// TIA Portal project "THESIS SCADA" (V15)

(* hardware
DEVICE "PC-System_1"  SIMATIC PC station
   slot 0: "SIMATIC PC station"  Rail  SIMATIC PC-Station  V1.0
      slot 125: "Stationmanager"  Station_Manager  V6.0.4
   slot 1: "HMI_RT_1"  WinCC RT Advanced  6AV2 104-0xxxx-xxxx  15.0.0.0
      slot 33792: "Host interface"  Host interface
*)

(* ===== HMI "HMI_RT_1" =====
system functions are stored by id; their names below are inferred from use
connection "Connection_1": OPC, OPC

HMI tags "Default tag table"
   "E1ALARM" : VT_I2, 1 s
   "E2ALARM" : VT_I2, 1 s
   "E3ALARM" : VT_I2, 1 s
   "E4ALARM" : VT_I2, 1 s
   "E1CAR" : VT_BOOL, 1 s
   "E2CAR" : VT_BOOL, 1 s
   "E3CAR" : VT_BOOL, 1 s
   "E4CAR" : VT_BOOL, 1 s
   "H0UP" : VT_BOOL, 1 s
   "H0DOWN" : VT_BOOL, 1 s
   "H1UP" : VT_BOOL, 1 s
   "H1DOWN" : VT_BOOL, 1 s
   "H2UP" : VT_BOOL, 1 s
   "H2DOWN" : VT_BOOL, 1 s
   "H3UP" : VT_BOOL, 1 s
   "H3DOWN" : VT_BOOL, 1 s
   "H4UP" : VT_BOOL, 1 s
   "H4DOWN" : VT_BOOL, 1 s
   "H5UP" : VT_BOOL, 1 s
   "H5DOWN" : VT_BOOL, 1 s
   "H6UP" : VT_BOOL, 1 s
   "H6DOWN" : VT_BOOL, 1 s
   "H7UP" : VT_BOOL, 1 s
   "H7DOWN" : VT_BOOL, 1 s
   "H8UP" : VT_BOOL, 1 s
   "H8DOWN" : VT_BOOL, 1 s
   "H9UP" : VT_BOOL, 1 s
   "H9DOWN" : VT_BOOL, 1 s
   "H10UP" : VT_BOOL, 1 s
   "H10DOWN" : VT_BOOL, 1 s
   "H11UP" : VT_BOOL, 1 s
   "H11DOWN" : VT_BOOL, 1 s
   "H12UP" : VT_BOOL, 1 s
   "H12DOWN" : VT_BOOL, 1 s
   "H13UP" : VT_BOOL, 1 s
   "H13DOWN" : VT_BOOL, 1 s
   "H14UP" : VT_BOOL, 1 s
   "H14DOWN" : VT_BOOL, 1 s
   "H15UP" : VT_BOOL, 1 s
   "H16DOWN" : VT_BOOL, 1 s
   "H17UP" : VT_BOOL, 1 s
   "H17DOWN" : VT_BOOL, 1 s
   "H18UP" : VT_BOOL, 1 s
   "H18DOWN" : VT_BOOL, 1 s
   "H19UP" : VT_BOOL, 1 s
   "H19DOWN" : VT_BOOL, 1 s
   "E1FLOOR0" : VT_BOOL, 1 s
   "E1FLOOR1" : VT_BOOL, 1 s
   "E1FLOOR2" : VT_BOOL, 1 s
   "E1FLOOR3" : VT_BOOL, 1 s
   "E1FLOOR4" : VT_BOOL, 1 s
   "E1FLOOR5" : VT_BOOL, 1 s
   "E1FLOOR6" : VT_BOOL, 1 s
   "E1FLOOR7" : VT_BOOL, 1 s
   "E1FLOOR8" : VT_BOOL, 1 s
   "E1FLOOR9" : VT_BOOL, 1 s
   "E1FLOOR10" : VT_BOOL, 1 s
   "E1FLOOR11" : VT_BOOL, 1 s
   "E1FLOOR12" : VT_BOOL, 1 s
   "E1FLOOR13" : VT_BOOL, 1 s
   "E2FLOOR0" : VT_BOOL, 1 s
   "E2FLOOR1" : VT_BOOL, 1 s
   "E2FLOOR2" : VT_BOOL, 1 s
   "E2FLOOR3" : VT_BOOL, 1 s
   "E2FLOOR4" : VT_BOOL, 1 s
   "E2FLOOR5" : VT_BOOL, 1 s
   "E2FLOOR6" : VT_BOOL, 1 s
   "E2FLOOR7" : VT_BOOL, 1 s
   "E2FLOOR8" : VT_BOOL, 1 s
   "E2FLOOR9" : VT_BOOL, 1 s
   "E2FLOOR10" : VT_BOOL, 1 s
   "E2FLOOR11" : VT_BOOL, 1 s
   "E2FLOOR12" : VT_BOOL, 1 s
   "E2FLOOR13" : VT_BOOL, 1 s
   "E3FLOOR0" : VT_BOOL, 1 s
   "E3FLOOR1" : VT_BOOL, 1 s
   "E3FLOOR2" : VT_BOOL, 1 s
   "E3FLOOR3" : VT_BOOL, 1 s
   "E3FLOOR4" : VT_BOOL, 1 s
   "E3FLOOR5" : VT_BOOL, 1 s
   "E3FLOOR6" : VT_BOOL, 1 s
   "E3FLOOR7" : VT_BOOL, 1 s
   "E3FLOOR8" : VT_BOOL, 1 s
   "E3FLOOR9" : VT_BOOL, 1 s
   "E3FLOOR10" : VT_BOOL, 1 s
   "E3FLOOR11" : VT_BOOL, 1 s
   "E3FLOOR12" : VT_BOOL, 1 s
   "E3FLOOR13" : VT_BOOL, 1 s
   "E4FLOOR5" : VT_BOOL, 1 s
   "E4FLOOR6" : VT_BOOL, 1 s
   "E4FLOOR7" : VT_BOOL, 1 s
   "E4FLOOR8" : VT_BOOL, 1 s
   "E4FLOOR9" : VT_BOOL, 1 s
   "E4FLOOR10" : VT_BOOL, 1 s
   "E4FLOOR11" : VT_BOOL, 1 s
   "E4FLOOR12" : VT_BOOL, 1 s
   "E4FLOOR13" : VT_BOOL, 1 s
   "E4FLOOR14" : VT_BOOL, 1 s
   "E4FLOOR15" : VT_BOOL, 1 s
   "E4FLOOR16" : VT_BOOL, 1 s
   "E4FLOOR17" : VT_BOOL, 1 s
   "E4FLOOR18" : VT_BOOL, 1 s
   "E4FLOOR19" : VT_BOOL, 1 s
   "E1CURRENTFLOOR" : VT_I2, 1 s
   "E2CURRENTFLOOR" : VT_I2, 1 s
   "E3CURRENTFLOOR" : VT_I2, 1 s
   "E4CURRENTFLOOR" : VT_I2, 1 s
   "E1UP" : VT_BOOL, 1 s
   "E1DOWN" : VT_BOOL, 1 s
   "E2UP" : VT_BOOL, 1 s
   "E2DOWN" : VT_BOOL, 1 s
   "E3UP" : VT_BOOL, 1 s
   "E3DOWN" : VT_BOOL, 1 s
   "E4UP" : VT_BOOL, 1 s
   "E4DOWN" : VT_BOOL, 1 s
   "ALARMRESET" : VT_BOOL, 1 s
   "ALARMNOT/RST" : VT_BOOL, 1 s
   "H16UP" : VT_BOOL, 1 s
   "H15DOWN" : VT_BOOL, 1 s
   "e1nextfloor" : VT_I2, 1 s
   "e2nextfloor" : VT_I2, 1 s
   "e3nextfloor" : VT_I2, 1 s
   "e4nextfloor" : VT_I2, 1 s

discrete alarms
   1: 'PLEASE GIVE CARCALL IN RESPECTIVE ELEVATOR DIRECTION', class Errors, trigger "E1ALARM" bit 0
   2: 'PLEASE GIVE CARCALL IN RESPECTIVE ELEVATOR DIRECTION', class Errors, trigger "E2ALARM" bit 0
   3: 'PLEASE GIVE CARCALL IN RESPECTIVE ELEVATOR DIRECTION', class Errors, trigger "E3ALARM" bit 0
   4: 'PLEASE GIVE CARCALL IN RESPECTIVE ELEVATOR DIRECTION', class Errors, trigger "E4ALARM" bit 0

screen "HALLCALL" 800x600
   TextField "Text field_1" at 208,16 size 148x37; Text 'HALLCALL'
   TextField "Text field_22" at 624,8 size 139x28; Text 'NAVIGATION'
   TextField "Text field_23" at 624,96 size 135x22; Text 'CURRENT FLOOR'
   TextField "Text field_24" at 624,208 size 135x22; Text 'CURRENT FLOOR'
   TextField "Text field_25" at 624,320 size 135x22; Text 'CURRENT FLOOR'
   TextField "Text field_26" at 632,432 size 135x22; Text 'CURRENT FLOOR'
   Group "Group_1" at 32,72 size 496x504
   Group "Group_2" at 648,544 size 96x31
   Group "Group_3" at 648,544 size 96x39
   Group "Group_4" at 648,544 size 96x40
   Group "Group_5" at 648,544 size 96x40
   Group "Group_6" at 648,544 size 96x40
   Group "Group_7" at 648,544 size 96x40
   Group "Group_8" at 648,544 size 96x40
   Group "Group_9" at 648,544 size 96x40
   Button "Button_1" at 640,280 size 96x32; TextOff 'E3CAR'
      on Click: ActivateScreen("E3CAR", 0)
   Button "Button_2" at 640,392 size 96x32; TextOff 'E4CAR'
      on Click: ActivateScreen("E4CAR", 0)
   Button "Button_3" at 640,168 size 96x32; TextOff 'E2CAR'
      on Click: ActivateScreen("E2CAR", 0)
   Button "Button_4" at 640,56 size 96x32; TextOff 'E1CAR'
      on Click: ActivateScreen("E1CAR", 0)
      Appearance <- "E1CAR"
   Button "Button_5" at 648,504 size 96x32; TextOff 'ALARM'
      on Click: ActivateScreen("ALARM", 0)
   IOField "I/O field_1" at 672,128 size 40x32; FormatPattern 11
      ProcessValue <- "E1CURRENTFLOOR"
   IOField "I/O field_2" at 672,240 size 40x32; FormatPattern 11
      ProcessValue <- "E2CURRENTFLOOR"
   IOField "I/O field_3" at 672,352 size 40x32; FormatPattern 11
      ProcessValue <- "E3CURRENTFLOOR"
   IOField "I/O field_4" at 672,464 size 40x32; FormatPattern 11
      ProcessValue <- "E4CURRENTFLOOR"
   Button "Button_24" at 48,94 size 96x32; TextOff 'H9UP'
      on Press: SetBit("H9UP")
      Appearance <- "H9UP"
   TextField "Text field_11" at 145,100 size 15x22; Text '9'
   Button "Button_25" at 161,94 size 96x32; TextOff 'H9DOWN'
      on Press: SetBit("H9DOWN")
      Appearance <- "H9DOWN"
   Button "Button_22" at 48,142 size 96x32; TextOff 'H8UP'
      on Press: SetBit("H8UP")
      Appearance <- "H8UP"
   TextField "Text field_10" at 145,148 size 15x22; Text '8'
   Button "Button_23" at 161,142 size 96x32; TextOff 'H8DOWN'
      on Press: SetBit("H8DOWN")
      Appearance <- "H8DOWN"
   Button "Button_20" at 48,190 size 96x32; TextOff 'H7UP'
      on Press: SetBit("H7UP")
      Appearance <- "H7UP"
   TextField "Text field_9" at 145,196 size 15x22; Text '7'
   Button "Button_21" at 161,190 size 96x32; TextOff 'H7DOWN'
      on Press: SetBit("H7DOWN")
      Appearance <- "H7DOWN"
   Button "Button_18" at 48,238 size 96x32; TextOff 'H6UP'
      on Press: SetBit("H6UP")
      Appearance <- "H6UP"
   TextField "Text field_8" at 145,244 size 15x22; Text '6'
   Button "Button_19" at 161,238 size 96x32; TextOff 'H6DOWN'
      on Press: SetBit("H6DOWN")
      Appearance <- "H0DOWN"
   Button "Button_16" at 48,286 size 96x32; TextOff 'H5UP'
      on Press: SetBit("H5UP")
      Appearance <- "H5UP"
   TextField "Text field_7" at 145,292 size 15x22; Text '5'
   Button "Button_17" at 161,286 size 96x32; TextOff 'H5DOWN'
      on Press: SetBit("H5DOWN")
      Appearance <- "H5DOWN"
   Button "Button_14" at 48,334 size 96x32; TextOff 'H4UP'
      on Press: SetBit("H4UP")
      Appearance <- "H4UP"
   TextField "Text field_6" at 145,340 size 15x22; Text '4'
   Button "Button_15" at 161,334 size 96x32; TextOff 'H4DOWN'
      on Press: SetBit("H4DOWN")
      Appearance <- "H4DOWN"
   Button "Button_12" at 48,382 size 96x32; TextOff 'H3UP'
      on Press: SetBit("H3UP")
      Appearance <- "H3UP"
   TextField "Text field_5" at 145,388 size 15x22; Text '3'
   Button "Button_13" at 161,382 size 96x32; TextOff 'H3DOWN'
      on Press: SetBit("H3DOWN")
      Appearance <- "H3DOWN"
   Button "Button_10" at 48,430 size 96x32; TextOff 'H2UP'
      on Press: SetBit("H2UP")
      Appearance <- "H2UP"
   TextField "Text field_4" at 145,436 size 15x22; Text '2'
   Button "Button_11" at 161,430 size 96x32; TextOff 'H2DOWN'
      on Press: SetBit("H2DOWN")
      Appearance <- "H2DOWN"
   Button "Button_8" at 48,478 size 96x32; TextOff 'H1UP'
      on Press: SetBit("H1UP")
      Appearance <- "H1UP"
   TextField "Text field_3" at 145,484 size 15x22; Text '1'
   Button "Button_9" at 161,478 size 96x32; TextOff 'H1DOWN'
      on Press: SetBit("H1DOWN")
      Appearance <- "H1DOWN"
   Button "Button_6" at 48,526 size 96x32; TextOff 'H0UP'
      on Press: SetBit("H0UP")
      Appearance <- "H0UP"
   TextField "Text field_2" at 145,532 size 15x22; Text '0'
   Button "Button_7" at 161,526 size 96x32; TextOff 'H0DOWN'
      on Press: SetBit("H0DOWN")
      Appearance <- "H0DOWN"
   Button "Button_44" at 288,94 size 96x32; TextOff 'H19UP'
      on Press: SetBit("H19UP")
      Appearance <- "H19UP"
   TextField "Text field_21" at 385,100 size 25x22; Text '19'
   Button "Button_45" at 410,93 size 96x32; TextOff 'H19DOWN'
      on Press: SetBit("H19DOWN")
      Appearance <- "H19DOWN"
   Button "Button_42" at 288,142 size 96x32; TextOff 'H18UP'
      on Press: SetBit("H18UP")
      Appearance <- "H18UP"
   TextField "Text field_20" at 385,148 size 25x22; Text '18'
   Button "Button_43" at 410,141 size 96x32; TextOff 'H18DOWN'
      on Press: SetBit("H18DOWN")
      Appearance <- "H18DOWN"
   Button "Button_40" at 288,190 size 96x32; TextOff 'H17UP'
      on Press: SetBit("H17UP")
      Appearance <- "H17UP"
   TextField "Text field_19" at 385,196 size 25x22; Text '17'
   Button "Button_41" at 410,189 size 96x32; TextOff 'H17DOWN'
      on Press: SetBit("H17DOWN")
      Appearance <- "H17DOWN"
   Button "Button_38" at 288,238 size 96x32; TextOff 'H16UP'
      on Press: SetBit("H16UP")
      Appearance <- "H16UP"
   TextField "Text field_18" at 385,244 size 25x22; Text '16'
   Button "Button_39" at 410,237 size 96x32; TextOff 'H16DOWN'
      on Press: SetBit("H16DOWN")
      Appearance <- "H16DOWN"
   Button "Button_36" at 288,286 size 96x32; TextOff 'H15UP'
      on Press: SetBit("H15UP")
      Appearance <- "H15UP"
   TextField "Text field_17" at 385,292 size 25x22; Text '15'
   Button "Button_37" at 410,285 size 96x32; TextOff 'H15DOWN'
      on Press: SetBit("H15DOWN")
      Appearance <- "H15DOWN"
   Button "Button_34" at 288,334 size 96x32; TextOff 'H14UP'
      on Press: SetBit("H14UP")
      Appearance <- "H14UP"
   TextField "Text field_16" at 385,340 size 25x22; Text '14'
   Button "Button_35" at 410,333 size 96x32; TextOff 'H14DOWN'
      on Press: SetBit("H14DOWN")
      Appearance <- "H14DOWN"
   Button "Button_32" at 288,382 size 96x32; TextOff 'H13UP'
      on Press: SetBit("H13UP")
      Appearance <- "H13UP"
   TextField "Text field_15" at 385,388 size 25x22; Text '13'
   Button "Button_33" at 410,381 size 96x32; TextOff 'H13DOWN'
      on Press: SetBit("H13DOWN")
      Appearance <- "H13DOWN"
   Button "Button_30" at 288,430 size 96x32; TextOff 'H12UP'
      on Press: SetBit("H12UP")
      Appearance <- "H12UP"
   TextField "Text field_14" at 385,436 size 25x22; Text '12'
   Button "Button_31" at 410,429 size 96x32; TextOff 'H12DOWN'
      on Press: SetBit("H12DOWN")
      Appearance <- "H12DOWN"
   Button "Button_28" at 288,478 size 96x32; TextOff 'H11UP'
      on Press: SetBit("H11UP")
      Appearance <- "H11UP"
   TextField "Text field_13" at 385,484 size 25x22; Text '11'
   Button "Button_29" at 410,477 size 96x32; TextOff 'H11DOWN'
      on Press: SetBit("H11DOWN")
      Appearance <- "H11DOWN"
   Button "Button_26" at 288,526 size 96x32; TextOff 'H10UP'
      on Press: SetBit("H10UP")
      Appearance <- "H10UP"
   TextField "Text field_12" at 385,532 size 25x22; Text '10'
   Button "Button_27" at 410,525 size 96x32; TextOff 'H10DOWN'
      on Press: SetBit("H10DOWN")
      Appearance <- "H10DOWN"
   TextField "Text field_27" at 651,552 size 86x22; Text 'NO ALARM'
   Rectangle "Rectangle_24" at 648,544 size 96x39
      Visibility <- "E4ALARM"
   TextField "Text field_28" at 655,555 size 81x22; Text 'E4 ALARM'
      Visibility <- "E4ALARM"
   TextField "Text field_29" at 651,554 size 86x22; Text 'NO ALARM'
   Rectangle "Rectangle_26" at 648,544 size 96x40
      Visibility <- "E3ALARM"
   TextField "Text field_30" at 655,555 size 81x22; Text 'E3 ALARM'
      Visibility <- "E3ALARM"
   TextField "Text field_31" at 651,554 size 86x22; Text 'NO ALARM'
   Rectangle "Rectangle_28" at 648,544 size 96x40
      Visibility <- "E2ALARM"
   TextField "Text field_32" at 655,555 size 81x22; Text 'E2 ALARM'
      Visibility <- "E2ALARM"
   TextField "Text field_33" at 651,554 size 86x22; Text 'NO ALARM'
   Rectangle "Rectangle_30" at 648,544 size 96x40
      Visibility <- "E1ALARM"
   TextField "Text field_34" at 655,555 size 81x22; Text 'E1 ALARM'
      Visibility <- "E1ALARM"

screen "E1CAR" 800x600
   TextField "Text field_1" at 659,516 size 86x22; Text 'NO ALARM'
   Group "Group" at 656,504 size 89x48
   Group "Group_1" at 648,504 size 96x48
   Button "Button_23" at 648,312 size 96x32; TextOff 'E2CAR'
      on Click: ActivateScreen("E2CAR", 0)
   Button "Button_24" at 648,360 size 96x32; TextOff 'E3CAR'
      on Click: ActivateScreen("E3CAR", 0)
   Button "Button_25" at 648,408 size 96x32; TextOff 'E4CAR'
      on Click: ActivateScreen("E4CAR", 0)
   Button "Button_26" at 648,456 size 96x32; TextOff 'ALARM'
      on Click: ActivateScreen("ALARM", 0)
   Rectangle "Rectangle_2" at 648,504 size 96x48
      Visibility <- "E1ALARM"
   TextField "Text field_2" at 655,517 size 81x22; Text 'E1 ALARM'
      Visibility <- "E1ALARM"
   TextField "Text field_3" at 16,8 size 167x37; Text 'E1 CARCALL'
   Rectangle "Rectangle_3" at 272,16 size 276x557
      Appearance <- "E1CAR"
   IOField "I/O field_1" at 360,176 size 104x32; FormatPattern 11
      ProcessValue <- "E1CURRENTFLOOR"
   Polyline "Polyline_2" at 368,72 size 32x40
      Appearance <- "E1UP"
   Polyline "Polyline_3" at 432,72 size 32x40
      Appearance <- "E1DOWN"
   IOField "I/O field_2" at 360,528 size 104x32; FormatPattern 99
      ProcessValue <- "e1nextfloor"
   TextField "Text field_4" at 328,32 size 176x22; Text 'ELEVATOR DIRECTION'
   TextField "Text field_5" at 344,144 size 135x22; Text 'CURRENT FLOOR'
   TextField "Text field_6" at 368,224 size 78x22; Text 'CAR CALL'
   TextField "Text field_7" at 328,496 size 176x22; Text 'NEXT SERVING FLOOR'
   Rectangle "Rectangle_4" at 360,256 size 104x232
      Appearance <- "E1CAR"
   Button "Button_1" at 368,360 size 24x24; TextOff '9'
      on Press: SetBit("E1FLOOR9")
      Appearance <- "E1FLOOR9"
   Button "Button_2" at 368,456 size 24x24; TextOff '18'
   Button "Button_3" at 368,392 size 24x24; TextOff '12'
      on Press: SetBit("E1FLOOR11")
      Appearance <- "E1FLOOR12"
   Button "Button_4" at 368,424 size 24x24; TextOff '15'
   Button "Button_5" at 400,360 size 24x24; TextOff '10'
      on Press: SetBit("E1FLOOR10")
      Appearance <- "E1FLOOR10"
   Button "Button_6" at 400,392 size 24x24; TextOff '13'
      Appearance <- "E1FLOOR13"
      on Press: SetBit("E1FLOOR13")
   Button "Button_7" at 400,456 size 24x24; TextOff '19'
   Button "Button_8" at 400,424 size 24x24; TextOff '16'
   Button "Button_9" at 432,264 size 24x24; TextOff '2'
      on Press: SetBit("E1FLOOR2")
      Appearance <- "E1FLOOR2"
   Button "Button_10" at 368,328 size 24x24; TextOff '6'
      on Press: SetBit("E1FLOOR6")
      Appearance <- "E1FLOOR6"
   Button "Button_11" at 400,328 size 24x24; TextOff '7'
      Appearance <- "E1FLOOR7"
      on Press: SetBit("E1FLOOR7")
   Button "Button_12" at 400,296 size 24x24; TextOff '4'
      Appearance <- "E1FLOOR4"
      on Press: SetBit("E1FLOOR4")
   Button "Button_13" at 368,296 size 24x24; TextOff '3'
      on Press: SetBit("E1FLOOR3")
      Appearance <- "E1FLOOR3"
   Button "Button_14" at 400,264 size 24x24; TextOff '1'
      on Press: SetBit("E1FLOOR1")
      Appearance <- "E1FLOOR1"
   Button "Button_15" at 368,264 size 24x24; TextOff '0'
      on Press: SetBit("E1FLOOR0")
      Appearance <- "E1FLOOR0"
   Button "Button_16" at 432,296 size 24x24; TextOff '5'
      on Press: SetBit("E1FLOOR5")
      Appearance <- "E1FLOOR5"
   Button "Button_17" at 432,328 size 24x24; TextOff '8'
      Appearance <- "E1FLOOR8"
      on Press: SetBit("E1FLOOR8")
   Button "Button_18" at 432,360 size 24x24; TextOff '11'
      Appearance <- "E1FLOOR11"
      on Press: SetBit("E1FLOOR11")
   Button "Button_19" at 432,392 size 24x24; TextOff '14'
   Button "Button_20" at 432,424 size 24x24; TextOff '17'
   Button "Button_21" at 432,456 size 24x24; TextOff 'Text'
   Group "Group_2" at 648,312 size 97x240
   TextField "Text field_22" at 624,240 size 139x28; Text 'NAVIGATION'

screen "E2CAR" 800x600
   Rectangle "Rectangle_2" at 648,504 size 96x48
      Visibility <- "E2ALARM"
   TextField "Text field_2" at 655,517 size 81x22; Text 'E2 ALARM'
      Visibility <- "E2ALARM"
   TextField "Text field_1" at 651,516 size 86x22; Text 'NO ALARM'
   Group "Group" at 648,504 size 96x48
   Group "Group_1" at 648,504 size 96x48
   TextField "Text field_3" at 12,19 size 167x37; Text 'E2 CARCALL'
   TextField "Text field_4" at 0,0 size 15x22; Text 'Text'
   Rectangle "Rectangle_6" at 272,16 size 276x557
      Appearance <- "E1CAR"
   IOField "I/O field_1" at 360,176 size 104x32; FormatPattern 11
      ProcessValue <- "E2CURRENTFLOOR"
   Polyline "Polyline_2" at 368,72 size 32x40
      Appearance <- "E2UP"
   Polyline "Polyline_3" at 432,72 size 32x40
      Appearance <- "E2DOWN"
   IOField "I/O field_2" at 360,528 size 104x32; FormatPattern 99
      ProcessValue <- "e2nextfloor"
   TextField "Text field_8" at 328,32 size 176x22; Text 'ELEVATOR DIRECTION'
   TextField "Text field_9" at 344,144 size 135x22; Text 'CURRENT FLOOR'
   TextField "Text field_10" at 368,224 size 78x22; Text 'CAR CALL'
   TextField "Text field_11" at 328,496 size 176x22; Text 'NEXT SERVING FLOOR'
   Rectangle "Rectangle_8" at 360,256 size 104x232
      Appearance <- "E2CAR"
   Button "Button_1" at 368,360 size 24x24; TextOff '9'
      on Press: SetBit("E2FLOOR9")
      Appearance <- "E2FLOOR9"
   Button "Button_2" at 368,456 size 24x24; TextOff '18'
   Button "Button_3" at 368,392 size 24x24; TextOff '12'
      on Press: SetBit("E2FLOOR11")
      Appearance <- "E2FLOOR12"
   Button "Button_4" at 368,424 size 24x24; TextOff '15'
   Button "Button_5" at 400,360 size 24x24; TextOff '10'
      on Press: SetBit("E2FLOOR10")
      Appearance <- "E2FLOOR10"
   Button "Button_6" at 400,392 size 24x24; TextOff '13'
      on Press: SetBit("E2FLOOR13")
      Appearance <- "E2FLOOR13"
   Button "Button_7" at 400,456 size 24x24; TextOff '19'
   Button "Button_8" at 400,424 size 24x24; TextOff '16'
   Button "Button_9" at 432,264 size 24x24; TextOff '2'
      on Press: SetBit("E2FLOOR2")
      Appearance <- "E2FLOOR2"
   Button "Button_10" at 368,328 size 24x24; TextOff '6'
      on Press: SetBit("E2FLOOR6")
      Appearance <- "E2FLOOR6"
   Button "Button_11" at 400,328 size 24x24; TextOff '7'
      on Press: SetBit("E2FLOOR7")
      Appearance <- "E2FLOOR7"
   Button "Button_12" at 400,296 size 24x24; TextOff '4'
      on Press: SetBit("E2FLOOR4")
      Appearance <- "E2FLOOR4"
   Button "Button_13" at 368,296 size 24x24; TextOff '3'
      on Press: SetBit("E2FLOOR3")
      Appearance <- "E2FLOOR3"
   Button "Button_14" at 400,264 size 24x24; TextOff '1'
      on Press: SetBit("E2FLOOR1")
      Appearance <- "E2FLOOR1"
   Button "Button_15" at 368,264 size 24x24; TextOff '0'
      on Press: SetBit("E2FLOOR0")
      Appearance <- "E2FLOOR0"
   Button "Button_16" at 432,296 size 24x24; TextOff '5'
      on Press: SetBit("E2FLOOR5")
      Appearance <- "E2FLOOR5"
   Button "Button_17" at 432,328 size 24x24; TextOff '8'
      on Press: SetBit("E2FLOOR8")
      Appearance <- "E2FLOOR8"
   Button "Button_18" at 432,360 size 24x24; TextOff '11'
      on Press: SetBit("E2FLOOR11")
      Appearance <- "E2FLOOR11"
   Button "Button_19" at 432,392 size 24x24; TextOff '14'
   Button "Button_20" at 432,424 size 24x24; TextOff '17'
   Button "Button_21" at 432,456 size 24x24; TextOff 'Text'
   Button "Button_22" at 648,304 size 96x32; TextOff 'E1CAR'
      on Click: ActivateScreen("E1CAR", 0)
      Appearance <- "E1CAR"
   Button "Button_24" at 648,352 size 96x32; TextOff 'E3CAR'
      on Click: ActivateScreen("E3CAR", 0)
   Button "Button_25" at 648,408 size 96x32; TextOff 'E4CAR'
      on Click: ActivateScreen("E4CAR", 0)
   Button "Button_26" at 648,456 size 96x32; TextOff 'ALARM'
      on Click: ActivateScreen("ALARM", 0)
   TextField "Text field_22" at 624,240 size 139x28; Text 'NAVIGATION'

screen "E3CAR" 800x600
   Rectangle "Rectangle_2" at 648,504 size 96x48
      Visibility <- "E3ALARM"
   TextField "Text field_2" at 655,517 size 81x22; Text 'E3 ALARM'
      Visibility <- "E3ALARM"
   TextField "Text field_1" at 651,516 size 86x22; Text 'NO ALARM'
   Group "Group" at 648,504 size 96x48
   Group "Group_1" at 648,504 size 96x48
   TextField "Text field_3" at 11,24 size 167x37; Text 'E3 CARCALL'
   TextField "Text field_7" at 0,0 size 15x22; Text 'Text'
   Rectangle "Rectangle_6" at 272,16 size 276x557
      Appearance <- "E1CAR"
   IOField "I/O field_1" at 360,176 size 104x32; FormatPattern 11
      ProcessValue <- "E3CURRENTFLOOR"
   Polyline "Polyline_2" at 368,72 size 32x40
      Appearance <- "E3UP"
   Polyline "Polyline_3" at 432,72 size 32x40
      Appearance <- "E3DOWN"
   IOField "I/O field_2" at 360,528 size 104x32; FormatPattern 99
      ProcessValue <- "e3nextfloor"
   TextField "Text field_8" at 328,32 size 176x22; Text 'ELEVATOR DIRECTION'
   TextField "Text field_9" at 344,144 size 135x22; Text 'CURRENT FLOOR'
   TextField "Text field_10" at 368,224 size 78x22; Text 'CAR CALL'
   TextField "Text field_11" at 328,496 size 176x22; Text 'NEXT SERVING FLOOR'
   Rectangle "Rectangle_8" at 360,256 size 104x232
      Appearance <- "E3CAR"
   Button "Button_1" at 368,360 size 24x24; TextOff '9'
      on Press: SetBit("E3FLOOR9")
      Appearance <- "E3FLOOR9"
   Button "Button_2" at 368,456 size 24x24; TextOff '18'
   Button "Button_3" at 368,392 size 24x24; TextOff '12'
      on Press: SetBit("E3FLOOR11")
      Appearance <- "E3FLOOR12"
   Button "Button_4" at 368,424 size 24x24; TextOff '15'
   Button "Button_5" at 400,360 size 24x24; TextOff '10'
      on Press: SetBit("E3FLOOR10")
      Appearance <- "E3FLOOR10"
   Button "Button_6" at 400,392 size 24x24; TextOff '13'
      on Press: SetBit("E3FLOOR13")
      Appearance <- "E3FLOOR13"
   Button "Button_7" at 400,456 size 24x24; TextOff '19'
   Button "Button_8" at 400,424 size 24x24; TextOff '16'
   Button "Button_9" at 432,264 size 24x24; TextOff '2'
      on Press: SetBit("E3FLOOR2")
      Appearance <- "E3FLOOR2"
   Button "Button_10" at 368,328 size 24x24; TextOff '6'
      on Press: SetBit("E3FLOOR6")
      Appearance <- "E3FLOOR6"
   Button "Button_11" at 400,328 size 24x24; TextOff '7'
      on Press: SetBit("E3FLOOR7")
      Appearance <- "E3FLOOR7"
   Button "Button_12" at 400,296 size 24x24; TextOff '4'
      on Press: SetBit("E3FLOOR4")
      Appearance <- "E3FLOOR4"
   Button "Button_13" at 368,296 size 24x24; TextOff '3'
      on Press: SetBit("E3FLOOR3")
      Appearance <- "E3FLOOR3"
   Button "Button_14" at 400,264 size 24x24; TextOff '1'
      on Press: SetBit("E3FLOOR1")
      Appearance <- "E3FLOOR1"
   Button "Button_15" at 368,264 size 24x24; TextOff '0'
      on Press: SetBit("E3FLOOR0")
      Appearance <- "E3FLOOR0"
   Button "Button_16" at 432,296 size 24x24; TextOff '5'
      on Press: SetBit("E3FLOOR5")
      Appearance <- "E3FLOOR5"
   Button "Button_17" at 432,328 size 24x24; TextOff '8'
      on Press: SetBit("E3FLOOR8")
      Appearance <- "E3FLOOR8"
   Button "Button_18" at 432,360 size 24x24; TextOff '11'
      on Press: SetBit("E3FLOOR11")
      Appearance <- "E3FLOOR11"
   Button "Button_19" at 432,392 size 24x24; TextOff '14'
   Button "Button_20" at 432,424 size 24x24; TextOff '17'
   Button "Button_21" at 432,456 size 24x24; TextOff 'Text'
   Button "Button_22" at 648,304 size 96x32; TextOff 'E1CAR'
      on Click: ActivateScreen("E1CAR", 0)
      Appearance <- "E1CAR"
   Button "Button_23" at 648,352 size 96x32; TextOff 'E2CAR'
      on Click: ActivateScreen("E2CAR", 0)
   Button "Button_25" at 648,400 size 96x32; TextOff 'E4CAR'
      on Click: ActivateScreen("E4CAR", 0)
   Button "Button_26" at 648,456 size 96x32; TextOff 'ALARM'
      on Click: ActivateScreen("ALARM", 0)
   TextField "Text field_22" at 624,240 size 139x28; Text 'NAVIGATION'

screen "E4CAR" 800x600
   Rectangle "Rectangle_2" at 648,504 size 96x48
      Visibility <- "E4ALARM"
   TextField "Text field_2" at 655,517 size 81x22; Text 'E4 ALARM'
      Visibility <- "E4ALARM"
   TextField "Text field_1" at 651,516 size 86x22; Text 'NO ALARM'
   Group "Group" at 648,504 size 96x48
   Group "Group_1" at 648,504 size 96x48
   TextField "Text field_3" at 12,20 size 167x37; Text 'E4 CARCALL'
   TextField "Text field_7" at 0,0 size 15x22; Text 'Text'
   Rectangle "Rectangle_6" at 272,16 size 276x557
      Appearance <- "E1CAR"
   IOField "I/O field_1" at 360,176 size 104x32; FormatPattern 11
      ProcessValue <- "E4CURRENTFLOOR"
   Polyline "Polyline_2" at 368,72 size 32x40
      Appearance <- "E4UP"
   Polyline "Polyline_3" at 432,72 size 32x40
      Appearance <- "E4DOWN"
   IOField "I/O field_2" at 360,528 size 104x32; FormatPattern 99
      ProcessValue <- "e4nextfloor"
   TextField "Text field_8" at 328,32 size 176x22; Text 'ELEVATOR DIRECTION'
   TextField "Text field_9" at 344,144 size 135x22; Text 'CURRENT FLOOR'
   TextField "Text field_10" at 368,224 size 78x22; Text 'CAR CALL'
   TextField "Text field_11" at 328,496 size 176x22; Text 'NEXT SERVING FLOOR'
   Rectangle "Rectangle_8" at 360,256 size 104x232
      Appearance <- "E4CAR"
   Button "Button_1" at 368,360 size 24x24; TextOff '9'
      on Press: SetBit("E4FLOOR9")
      Appearance <- "E4FLOOR9"
   Button "Button_2" at 368,456 size 24x24; TextOff '18'
      on Press: SetBit("E4FLOOR18")
      Appearance <- "E4FLOOR18"
   Button "Button_3" at 368,392 size 24x24; TextOff '12'
      on Press: SetBit("E4FLOOR11")
      Appearance <- "E4FLOOR12"
   Button "Button_4" at 368,424 size 24x24; TextOff '15'
      on Press: SetBit("E4FLOOR15")
      Appearance <- "E4FLOOR15"
   Button "Button_5" at 400,360 size 24x24; TextOff '10'
      on Press: SetBit("E4FLOOR10")
      Appearance <- "E4FLOOR10"
   Button "Button_6" at 400,392 size 24x24; TextOff '13'
      on Press: SetBit("E4FLOOR13")
      Appearance <- "E4FLOOR13"
   Button "Button_7" at 400,456 size 24x24; TextOff '19'
      Appearance <- "E4FLOOR19"
      on Press: SetBit("E4FLOOR19")
   Button "Button_8" at 400,424 size 24x24; TextOff '16'
      on Press: SetBit("E4FLOOR16")
      Appearance <- "E4FLOOR16"
   Button "Button_9" at 432,264 size 24x24; TextOff '2'
      on Press: SetBit("E2FLOOR2")
      Appearance <- "E2FLOOR2"
   Button "Button_10" at 368,328 size 24x24; TextOff '6'
      on Press: SetBit("E4FLOOR6")
      Appearance <- "E4FLOOR6"
   Button "Button_11" at 400,328 size 24x24; TextOff '7'
      on Press: SetBit("E4FLOOR7")
      Appearance <- "E4FLOOR7"
   Button "Button_12" at 400,296 size 24x24; TextOff '4'
      on Press: SetBit("E2FLOOR4")
      Appearance <- "E2FLOOR4"
   Button "Button_13" at 368,296 size 24x24; TextOff '3'
      on Press: SetBit("E2FLOOR3")
      Appearance <- "E2FLOOR3"
   Button "Button_14" at 400,264 size 24x24; TextOff '1'
      on Press: SetBit("E2FLOOR1")
      Appearance <- "E2FLOOR1"
   Button "Button_15" at 368,264 size 24x24; TextOff '0'
      on Press: SetBit("E2FLOOR0")
      Appearance <- "E2FLOOR0"
   Button "Button_16" at 432,296 size 24x24; TextOff '5'
      on Press: SetBit("E4FLOOR5")
      Appearance <- "E4FLOOR5"
   Button "Button_17" at 432,328 size 24x24; TextOff '8'
      on Press: SetBit("E4FLOOR8")
      Appearance <- "E4FLOOR8"
   Button "Button_18" at 432,360 size 24x24; TextOff '11'
      on Press: SetBit("E4FLOOR11")
      Appearance <- "E4FLOOR11"
   Button "Button_19" at 432,392 size 24x24; TextOff '14'
      Appearance <- "E4FLOOR14"
      on Press: SetBit("E4FLOOR14")
   Button "Button_20" at 432,424 size 24x24; TextOff '17'
      on Press: SetBit("E4FLOOR17")
      Appearance <- "E4FLOOR17"
   Button "Button_21" at 432,456 size 24x24; TextOff 'Text'
   Button "Button_22" at 648,312 size 96x32; TextOff 'E1CAR'
      on Click: ActivateScreen("E1CAR", 0)
      Appearance <- "E1CAR"
   Button "Button_23" at 648,360 size 96x32; TextOff 'E2CAR'
      on Click: ActivateScreen("E2CAR", 0)
   Button "Button_24" at 648,408 size 96x32; TextOff 'E3CAR'
      on Click: ActivateScreen("E3CAR", 0)
   Button "Button_26" at 648,456 size 96x32; TextOff 'ALARM'
      on Click: ActivateScreen("ALARM", 0)
   TextField "Text field_22" at 624,240 size 139x28; Text 'NAVIGATION'

screen "ALARM" 800x600
   AlarmView "Alarm view_1" at 24,80 size 736x340
   Button "Button_22" at 56,536 size 96x32; TextOff 'E1CAR'
      on Click: ActivateScreen("E1CAR", 0)
      Appearance <- "E1CAR"
   Button "Button_23" at 192,536 size 96x32; TextOff 'E2CAR'
      on Click: ActivateScreen("E2CAR", 0)
   Button "Button_24" at 328,536 size 96x32; TextOff 'E3CAR'
      on Click: ActivateScreen("E3CAR", 0)
   Button "Button_25" at 464,536 size 96x32; TextOff 'E4CAR'
      on Click: ActivateScreen("E4CAR", 0)
   Button "Button_26" at 608,536 size 96x32; TextOff 'HALL CALL'
      on Click: ActivateScreen("HALLCALL", 0)
   TextField "Text field_3" at 304,16 size 104x37; Text 'ALARM'
   Button "Button_1" at 624,456 size 96x32; TextOff 'RESET'
      on Press: SetBit("ALARMRESET")
      on Release: ResetBit("ALARMRESET")
   Group "Group_2" at 96,448 size 96x31
   Group "Group_3" at 96,448 size 96x39
   Group "Group_4" at 96,448 size 96x40
   Group "Group_5" at 96,448 size 96x40
   Group "Group_6" at 96,448 size 96x40
   Group "Group_7" at 96,448 size 96x40
   Group "Group_8" at 96,448 size 96x40
   Group "Group_9" at 96,448 size 96x40
   TextField "Text field_27" at 99,456 size 86x22; Text 'NO ALARM'
   Rectangle "Rectangle_24" at 96,448 size 96x39
      Visibility <- "E4ALARM"
   TextField "Text field_28" at 103,459 size 81x22; Text 'E4 ALARM'
      Visibility <- "E4ALARM"
   TextField "Text field_29" at 99,458 size 86x22; Text 'NO ALARM'
   Rectangle "Rectangle_26" at 96,448 size 96x40
      Visibility <- "E3ALARM"
   TextField "Text field_30" at 103,459 size 81x22; Text 'E3 ALARM'
      Visibility <- "E3ALARM"
   TextField "Text field_31" at 99,458 size 86x22; Text 'NO ALARM'
   Rectangle "Rectangle_28" at 96,448 size 96x40
      Visibility <- "E2ALARM"
   TextField "Text field_32" at 103,459 size 81x22; Text 'E2 ALARM'
      Visibility <- "E2ALARM"
   TextField "Text field_33" at 99,458 size 86x22; Text 'NO ALARM'
   Rectangle "Rectangle_30" at 96,448 size 96x40
      Visibility <- "E1ALARM"
   TextField "Text field_34" at 103,459 size 81x22; Text 'E1 ALARM'
      Visibility <- "E1ALARM"
*)